FUNCTION_BLOCK AB2_BYTE_TO_B (* Composite FB for convert AYTE to AB2 *)
  (* Standard: 61499-2; Description: Copyright (c) 2024 HR Agrartechnik GmbH This program and the accompanying materials are made available under the terms of the Eclipse Public License 2.0 which is available at https://www.eclipse.org/legal/epl-2.0/ SPDX-License-Identifier: EPL-2.0 *)
  (* Version 1.0, 2024-04-24, Franz Höpfinger, HR Agrartechnik GmbH *)
  PACKAGE adapter::conversion::bidirectional;
  IMPORT eclipse4diac::core::TypeHash;
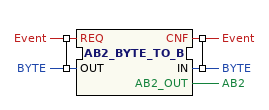
  EVENT_INPUT
    REQ WITH OUT; (* Request to Adapter *)
  END_EVENT
  EVENT_OUTPUT
    CNF WITH IN; (* Confirmation from Adapter *)
  END_EVENT
  VAR_INPUT
    OUT : BYTE; (* Output data to Adapter *)
  END_VAR
  VAR_OUTPUT
    IN : BYTE; (* Input data from Adapter *)
  END_VAR
  PLUGS
    AB2_OUT : adapter::types::bidirectional::AB2; (* Adapter Output *)
  END_PLUGS
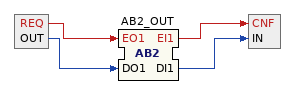
  EVENT_CONNECTIONS
    REQ TO AB2_OUT.EO1;
    AB2_OUT.EI1 TO CNF;
  END_CONNECTIONS
  DATA_CONNECTIONS
    OUT TO AB2_OUT.DO1;
    AB2_OUT.DI1 TO IN;
  END_CONNECTIONS
END_FUNCTION_BLOCK
